FUNCTION_BLOCK ST_CREATE_FB (* Creates a FB instance from a certain FB type *)
  (* Standard: 61499-1; Classification: Reconfiguration; Function: Creates FB or Resource instance; Type: Structural Service *)
  (* Version 1.0, 2012-05-31, EG, 4DIAC-Consortium *)
  (* Compiler Cpp GNU GCC >3.0 *)
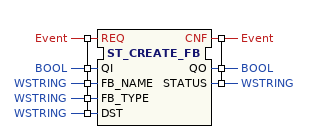
  EVENT_INPUT
    REQ WITH FB_NAME, FB_TYPE, DST, QI; (* Event to require creation of a FB or Resource instance *)
  END_EVENT
  EVENT_OUTPUT
    CNF WITH STATUS, QO; (* Event to confirm that the FB or Resource instance has been created *)
  END_EVENT
  VAR_INPUT
    QI : BOOL; (* Event Input Qualifier *)
    FB_NAME : WSTRING; (* Name of the FB instance *)
    FB_TYPE : WSTRING; (* FB type name *)
    DST : WSTRING; (* Destination where the FB or Resource instance has to be created (Syntax: ResourceName) *)
  END_VAR
  VAR_OUTPUT
    QO : BOOL; (* Event Output Qualifier *)
    STATUS : WSTRING; (* Service Status: RDY, UNSUPPORTED_TYPE, INVALID_OPERATION, INVALID_STATE *)
  END_VAR
  SERVICE APPLICATION/RESOURCE (* Creates a FB instance from a certain FB type *)
    SEQUENCE normal_establishment
      APPLICATION.INIT+() -> APPLICATION.INITO+();
    END_SEQUENCE
    SEQUENCE unsuccessful_establishment
      APPLICATION.INIT+() -> APPLICATION.INITO-();
    END_SEQUENCE
    SEQUENCE request_confirm
      APPLICATION.REQ+() -> APPLICATION.CNF+();
    END_SEQUENCE
    SEQUENCE request_inhibited
      APPLICATION.REQ-() -> APPLICATION.CNF-();
    END_SEQUENCE
    SEQUENCE request_error
      APPLICATION.REQ+() -> APPLICATION.CNF-();
    END_SEQUENCE
    SEQUENCE application_initiated_termination
      APPLICATION.INIT-() -> APPLICATION.INITO-();
    END_SEQUENCE
    SEQUENCE resource_initiated_termination
      -> APPLICATION.INITO-();
    END_SEQUENCE
  END_SERVICE
END_FUNCTION_BLOCK
